SUBAPPLICATION Uebung_018 (* Control Audio Signal und Delay *)
  (* Standard: 61499-2; Description: Copyright (c) 2023 Meisterschulen am Ostbahnhof This program and the accompanying materials are made available under the terms of the Eclipse Public License 2.0 which is available at https://www.eclipse.org/legal/epl-2.0/ SPDX-License-Identifier: EPL-2.0 *)
  (* Version 1.0, 2023-10-23, Franz Höpfinger, Meisterschulen am Ostbahnhof *)
  PACKAGE Uebungen;
  IMPORT SoftKeyActivationCode::SK_RELEASED;
  IMPORT Uebungen::const::UT::DefaultPool::SoftKey_F1;
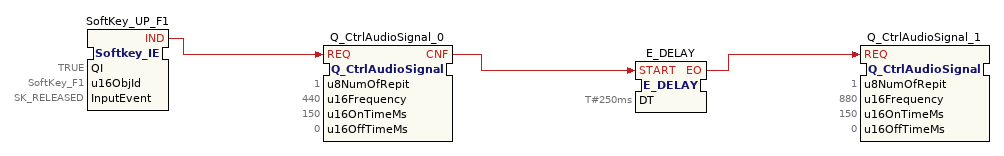
  FBS
    SoftKey_UP_F1 : Softkey_IE(QI := TRUE, u16ObjId := SoftKey_F1, InputEvent := SK_RELEASED);
    Q_CtrlAudioSignal_0 : isobus::ut::Q_CtrlAudioSignal(u8NumOfRepit := 1, u16Frequency := 440, u16OnTimeMs := 150, u16OffTimeMs := 0);
    Q_CtrlAudioSignal_1 : isobus::ut::Q_CtrlAudioSignal(u8NumOfRepit := 1, u16Frequency := 880, u16OnTimeMs := 150, u16OffTimeMs := 0);
    E_DELAY : iec61499::events::E_DELAY(DT := T#250ms);
  END_FBS
  EVENT_CONNECTIONS
    SoftKey_UP_F1.IND TO Q_CtrlAudioSignal_0.REQ;
    E_DELAY.EO TO Q_CtrlAudioSignal_1.REQ;
    Q_CtrlAudioSignal_0.CNF TO E_DELAY.START;
  END_CONNECTIONS
END_SUBAPPLICATION
